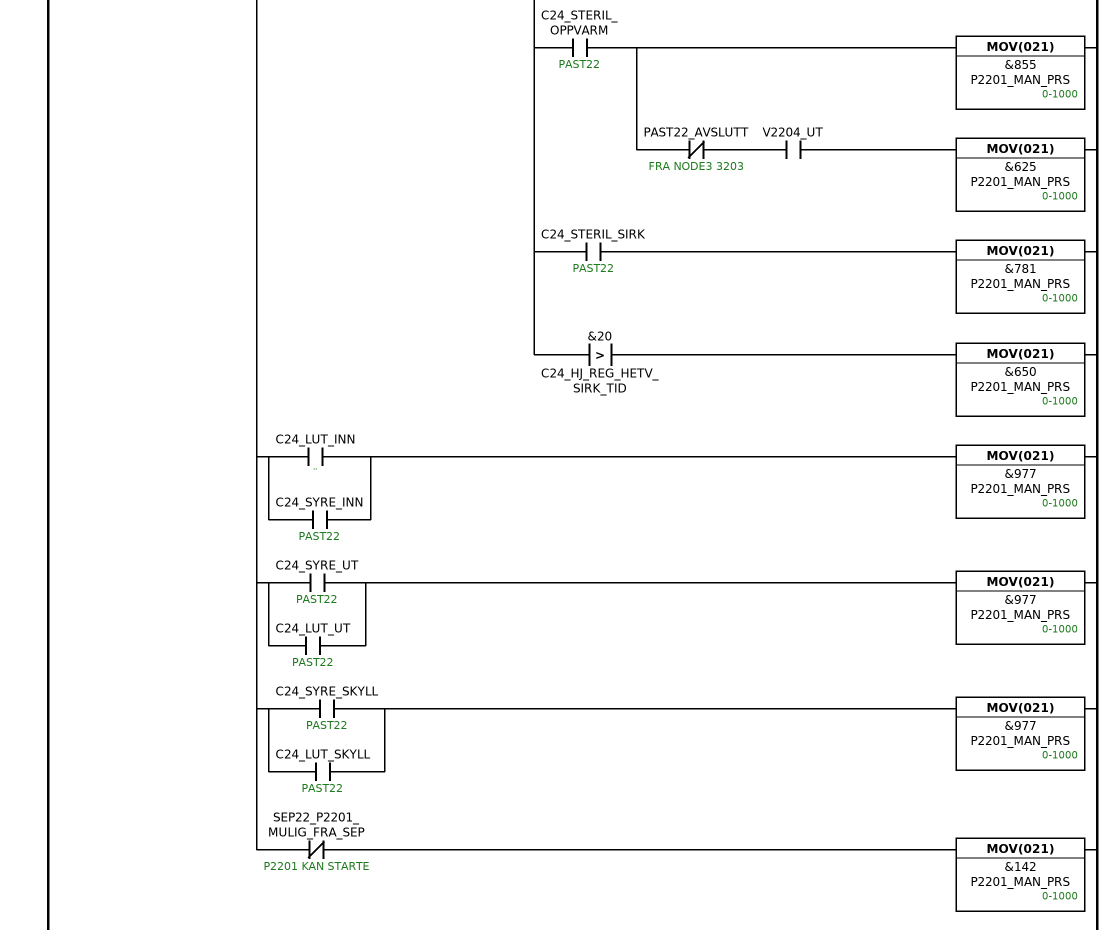
; [picture p1176: NewProgram1 / P2201, rungs 5-5]
; rung 5: REGULATOR P2201 MANUELT SETPUNKT I 0-1000
LD P_On
OUT TR0
ANDNOT PGM504_IND_C24  ; VASK PAST22
OUT TR1
AND SEP22_PART_SKUDD_INNE_FRA_SEP  ; SEP22 PARTIALSKUDD
ANDNOT 915.08
MOV(021) &590 P2201_MAN_PRS  ; 0-1000
LD TR1
AND 915.08
MOV(021) &0 P2201_MAN_PRS  ; 0-1000
LD TR0
AND PGM504_IND_C24  ; VASK PAST22
OUT TR0
@AND SEP22_PART_SKUDD_INNE_FRA_SEP  ; SEP22 PARTIALSKUDD
MOV(021) &590 P2201_MAN_PRS  ; 0-1000
LD TR0
@AND SEP22_TOT_SKUDD_INNE_FRA_SEP  ; SEP22 TOTALSKUDD(VASK)
OUT TR1
AND C24_FORSKYLL  ; PAST22
MOV(021) &448 P2201_MAN_PRS  ; 0-1000
LD TR1
AND C24_SYRE_SIRK  ; PAST22
MOV(021) &448 P2201_MAN_PRS  ; 0-1000
LD TR1
AND C24_LUT_SIRK  ; PAST22
MOV(021) &448 P2201_MAN_PRS  ; 0-1000
LD TR0
ANDNOT SEP22_PART_SKUDD_INNE_FRA_SEP  ; SEP22 PARTIALSKUDD
ANDNOT SEP22_TOT_SKUDD_INNE_FRA_SEP  ; SEP22 TOTALSKUDD(VASK)
OUT TR1
MOV(021) &977 P2201_MAN_PRS  ; 0-1000
ANDNOT PAST22_AVSLUTT  ; FRA NODE3 3203
AND V2204_UT
MOV(021) &977 P2201_MAN_PRS  ; 0-1000
LD TR1
AND C24_FORSKYLL  ; PAST22
MOV(021) &977 P2201_MAN_PRS  ; 0-1000
LD TR1
LD C24_SYRE_SIRK  ; PAST22
OR C24_LUT_SIRK  ; PAST22
ANDLD
MOV(021) &879 P2201_MAN_PRS  ; 0-1000
ANDNOT PAST22_AVSLUTT  ; FRA NODE3 3203
AND V2204_UT
MOV(021) &855 P2201_MAN_PRS  ; 0-1000
LD TR1
AND C24_STERIL_OPPVARM  ; PAST22
MOV(021) &855 P2201_MAN_PRS  ; 0-1000
ANDNOT PAST22_AVSLUTT  ; FRA NODE3 3203
AND V2204_UT
MOV(021) &625 P2201_MAN_PRS  ; 0-1000
LD TR1
AND C24_STERIL_SIRK  ; PAST22
MOV(021) &781 P2201_MAN_PRS  ; 0-1000
LD TR1
AND>(320) &20 C24_HJ_REG_HETV_SIRK_TID
MOV(021) &650 P2201_MAN_PRS  ; 0-1000
LD TR0
LD C24_LUT_INN  ; ¨
OR C24_SYRE_INN  ; PAST22
ANDLD
MOV(021) &977 P2201_MAN_PRS  ; 0-1000
LD TR0
LD C24_SYRE_UT  ; PAST22
OR C24_LUT_UT  ; PAST22
ANDLD
MOV(021) &977 P2201_MAN_PRS  ; 0-1000
LD TR0
LD C24_SYRE_SKYLL  ; PAST22
OR C24_LUT_SKYLL  ; PAST22
ANDLD
MOV(021) &977 P2201_MAN_PRS  ; 0-1000
LD TR0
ANDNOT SEP22_P2201_MULIG_FRA_SEP  ; P2201 KAN STARTE
MOV(021) &142 P2201_MAN_PRS  ; 0-1000

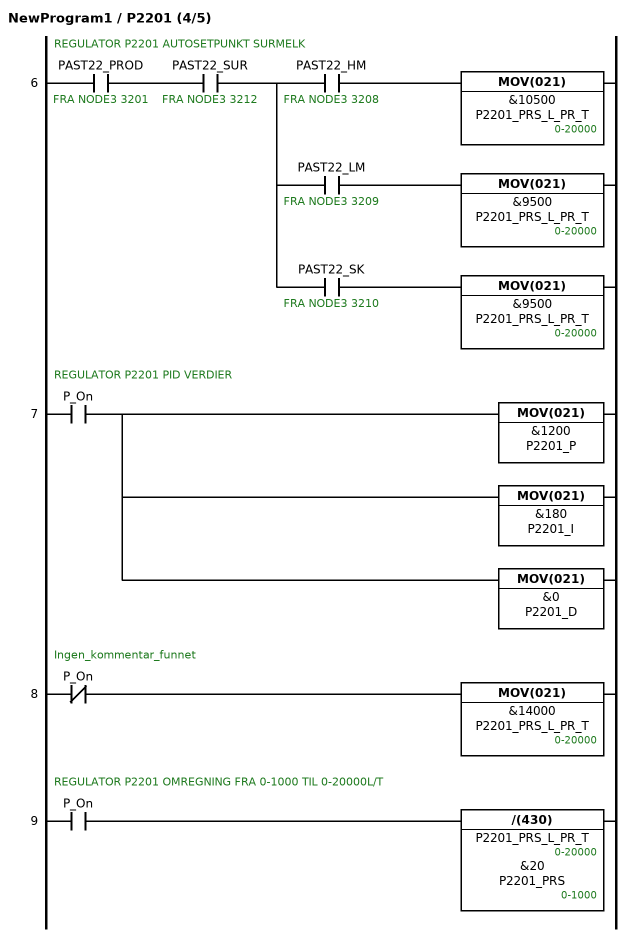
; rung 6: REGULATOR P2201 AUTOSETPUNKT SURMELK
LD PAST22_PROD  ; FRA NODE3 3201
AND PAST22_SUR  ; FRA NODE3 3212
OUT TR0
AND PAST22_HM  ; FRA NODE3 3208
MOV(021) &10500 P2201_PRS_L_PR_T  ; 0-20000
LD TR0
AND PAST22_LM  ; FRA NODE3 3209
MOV(021) &9500 P2201_PRS_L_PR_T  ; 0-20000
LD TR0
AND PAST22_SK  ; FRA NODE3 3210
MOV(021) &9500 P2201_PRS_L_PR_T  ; 0-20000
; rung 7: REGULATOR P2201 PID VERDIER
LD P_On
MOV(021) &1200 P2201_P
MOV(021) &180 P2201_I
MOV(021) &0 P2201_D
; rung 8: Ingen_kommentar_funnet
LDNOT P_On
MOV(021) &14000 P2201_PRS_L_PR_T  ; 0-20000
; rung 9: REGULATOR P2201 OMREGNING FRA 0-1000 TIL 0-20000L/T
LD P_On
/(430) P2201_PRS_L_PR_T &20 P2201_PRS  ; 0-20000, 0-1000

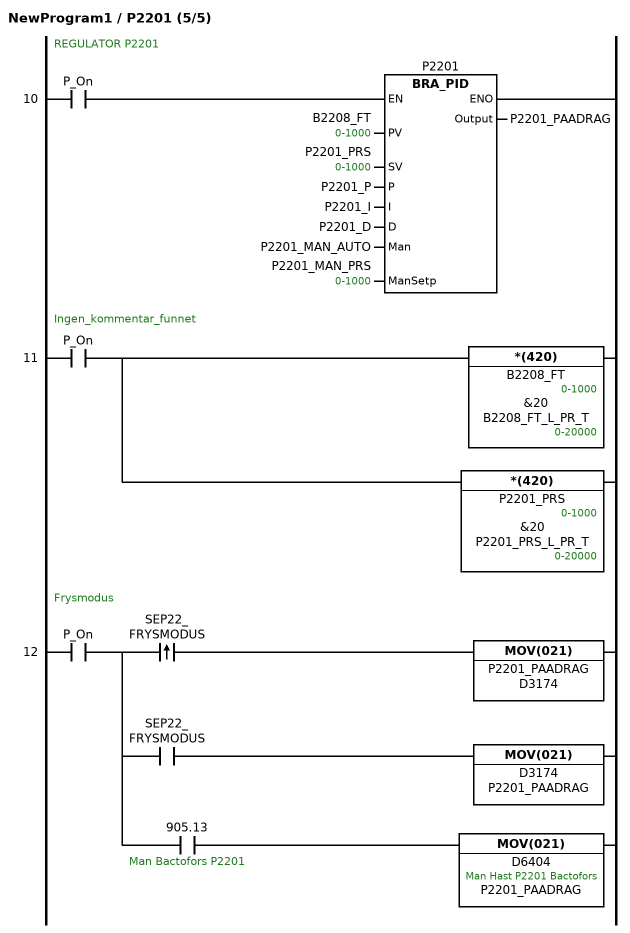
; rung 10: REGULATOR P2201
LD P_On
CALL P2201 : BRA_PID (PV := B2208_FT, SV := P2201_PRS, P := P2201_P, I := P2201_I, D := P2201_D, Man := P2201_MAN_AUTO, ManSetp := P2201_MAN_PRS, Output => P2201_PAADRAG)  ; 0-1000
; rung 11: Ingen_kommentar_funnet
LD P_On
*(420) B2208_FT &20 B2208_FT_L_PR_T  ; 0-1000, 0-20000
*(420) P2201_PRS &20 P2201_PRS_L_PR_T  ; 0-1000, 0-20000
; rung 12: Frysmodus
LD P_On
OUT TR0
@AND SEP22_FRYSMODUS
MOV(021) P2201_PAADRAG D3174
LD TR0
AND SEP22_FRYSMODUS
MOV(021) D3174 P2201_PAADRAG
LD TR0
AND 905.13  ; Man Bactofors P2201
MOV(021) D6404 P2201_PAADRAG  ; Man Hast P2201 Bactofors
; rung 13: Ingen_kommentar_funnet

### Section P2202

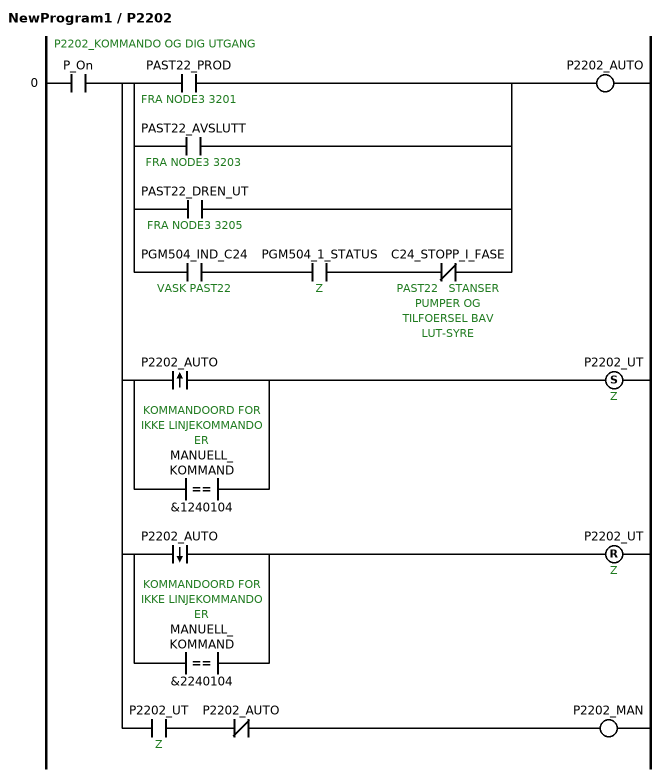
; rung 0: P2202_KOMMANDO OG DIG UTGANG
LD P_On
OUT TR0
LD PAST22_PROD  ; FRA NODE3 3201
OR PAST22_AVSLUTT  ; FRA NODE3 3203
OR PAST22_DREN_UT  ; FRA NODE3 3205
LD PGM504_IND_C24  ; VASK PAST22
AND PGM504_1_STATUS  ; Z
ANDNOT C24_STOPP_I_FASE  ; PAST22   STANSER PUMPER OG TILFOERSEL BAV LUT-SYRE
ORLD
ANDLD
OUT P2202_AUTO
LD TR0
@LD P2202_AUTO
OR=L(301) MANUELL_KOMMAND &1240104  ; KOMMANDOORD FOR IKKE LINJEKOMMANDOER
ANDLD
SET P2202_UT  ; Z
LD TR0
%LD P2202_AUTO
OR=L(301) MANUELL_KOMMAND &2240104  ; KOMMANDOORD FOR IKKE LINJEKOMMANDOER
ANDLD
RSET P2202_UT  ; Z
LD TR0
AND P2202_UT  ; Z
ANDNOT P2202_AUTO
OUT P2202_MAN
; rung 1: Ingen_kommentar_funnet

### Section P2203

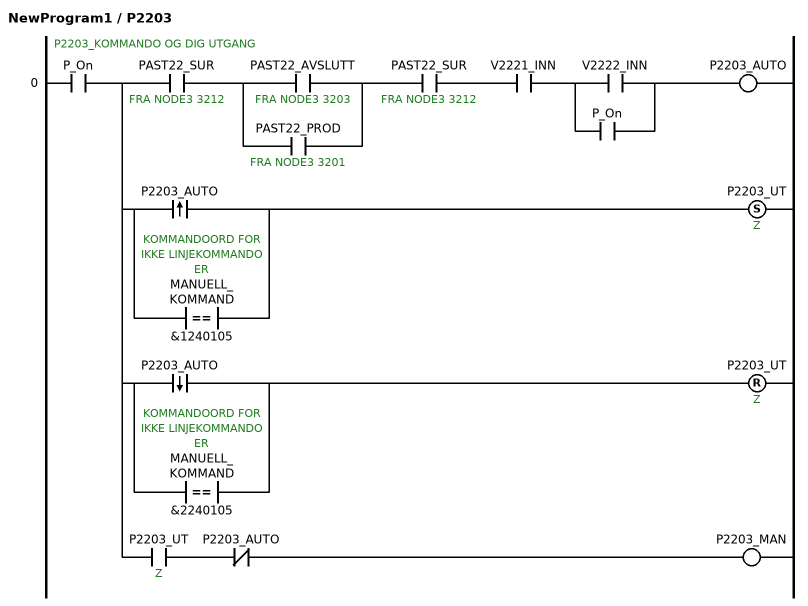
; rung 0: P2203_KOMMANDO OG DIG UTGANG
LD P_On
OUT TR0
AND PAST22_SUR  ; FRA NODE3 3212
LD PAST22_AVSLUTT  ; FRA NODE3 3203
OR PAST22_PROD  ; FRA NODE3 3201
ANDLD
AND PAST22_SUR  ; FRA NODE3 3212
AND V2221_INN
LD V2222_INN
OR P_On
ANDLD
OUT P2203_AUTO
LD TR0
@LD P2203_AUTO
OR=L(301) MANUELL_KOMMAND &1240105  ; KOMMANDOORD FOR IKKE LINJEKOMMANDOER
ANDLD
SET P2203_UT  ; Z
LD TR0
%LD P2203_AUTO
OR=L(301) MANUELL_KOMMAND &2240105  ; KOMMANDOORD FOR IKKE LINJEKOMMANDOER
ANDLD
RSET P2203_UT  ; Z
LD TR0
AND P2203_UT  ; Z
ANDNOT P2203_AUTO
OUT P2203_MAN
; rung 1: Ingen_kommentar_funnet

### Section P2204

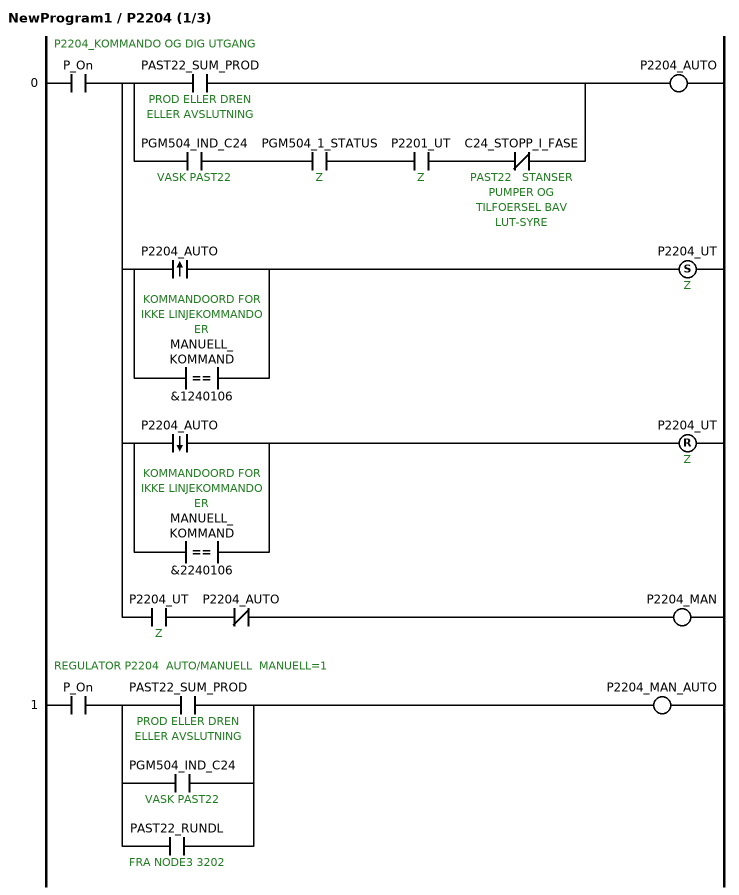
; rung 0: P2204_KOMMANDO OG DIG UTGANG
LD P_On
OUT TR0
LD PAST22_SUM_PROD  ; PROD ELLER DREN ELLER AVSLUTNING
LD PGM504_IND_C24  ; VASK PAST22
AND PGM504_1_STATUS  ; Z
AND P2201_UT  ; Z
ANDNOT C24_STOPP_I_FASE  ; PAST22   STANSER PUMPER OG TILFOERSEL BAV LUT-SYRE
ORLD
ANDLD
OUT P2204_AUTO
LD TR0
@LD P2204_AUTO
OR=L(301) MANUELL_KOMMAND &1240106  ; KOMMANDOORD FOR IKKE LINJEKOMMANDOER
ANDLD
SET P2204_UT  ; Z
LD TR0
%LD P2204_AUTO
OR=L(301) MANUELL_KOMMAND &2240106  ; KOMMANDOORD FOR IKKE LINJEKOMMANDOER
ANDLD
RSET P2204_UT  ; Z
LD TR0
AND P2204_UT  ; Z
ANDNOT P2204_AUTO
OUT P2204_MAN
; rung 1: REGULATOR P2204  AUTO/MANUELL  MANUELL=1
LD P_On
LD PAST22_SUM_PROD  ; PROD ELLER DREN ELLER AVSLUTNING
OR PGM504_IND_C24  ; VASK PAST22
OR PAST22_RUNDL  ; FRA NODE3 3202
ANDLD
OUT P2204_MAN_AUTO

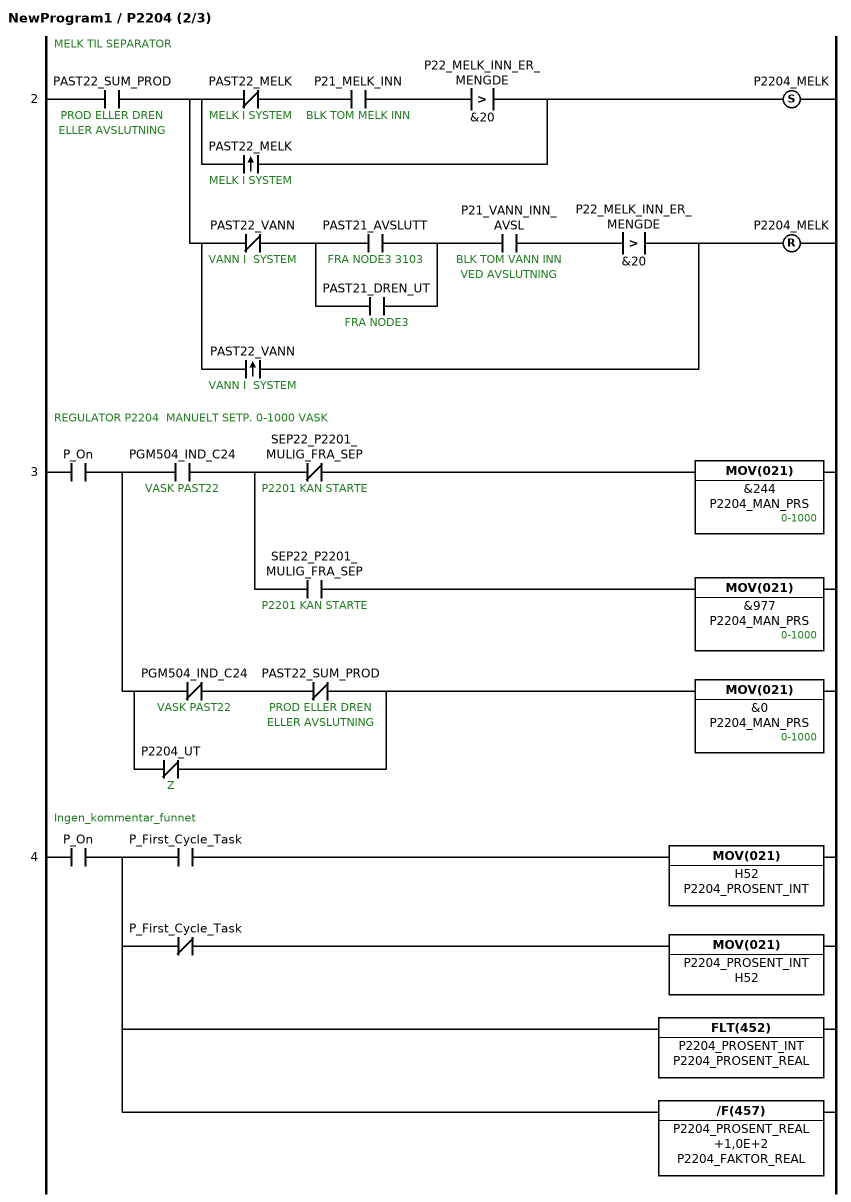
; rung 2: MELK TIL SEPARATOR
LD PAST22_SUM_PROD  ; PROD ELLER DREN ELLER AVSLUTNING
OUT TR0
LDNOT PAST22_MELK  ; MELK I SYSTEM
AND P21_MELK_INN  ; BLK TOM MELK INN
AND>L(321) P22_MELK_INN_ER_MENGDE &20
@OR PAST22_MELK  ; MELK I SYSTEM
ANDLD
SET P2204_MELK
LD TR0
LDNOT PAST22_VANN  ; VANN I  SYSTEM
LD PAST21_AVSLUTT  ; FRA NODE3 3103
OR PAST21_DREN_UT  ; FRA NODE3
ANDLD
AND P21_VANN_INN_AVSL  ; BLK TOM VANN INN VED AVSLUTNING
AND>L(321) P22_MELK_INN_ER_MENGDE &20
@OR PAST22_VANN  ; VANN I  SYSTEM
ANDLD
RSET P2204_MELK
; rung 3: REGULATOR P2204  MANUELT SETP. 0-1000 VASK
LD P_On
OUT TR0
AND PGM504_IND_C24  ; VASK PAST22
OUT TR1
ANDNOT SEP22_P2201_MULIG_FRA_SEP  ; P2201 KAN STARTE
MOV(021) &244 P2204_MAN_PRS  ; 0-1000
LD TR1
AND SEP22_P2201_MULIG_FRA_SEP  ; P2201 KAN STARTE
MOV(021) &977 P2204_MAN_PRS  ; 0-1000
LD TR0
LDNOT PGM504_IND_C24  ; VASK PAST22
ANDNOT PAST22_SUM_PROD  ; PROD ELLER DREN ELLER AVSLUTNING
ORNOT P2204_UT  ; Z
ANDLD
MOV(021) &0 P2204_MAN_PRS  ; 0-1000
; rung 4: Ingen_kommentar_funnet
LD P_On
OUT TR0
AND P_First_Cycle_Task
MOV(021) H52 P2204_PROSENT_INT
LD TR0
ANDNOT P_First_Cycle_Task
MOV(021) P2204_PROSENT_INT H52
LD TR0
FLT(452) P2204_PROSENT_INT P2204_PROSENT_REAL
/F(457) P2204_PROSENT_REAL +1,0E+2 P2204_FAKTOR_REAL

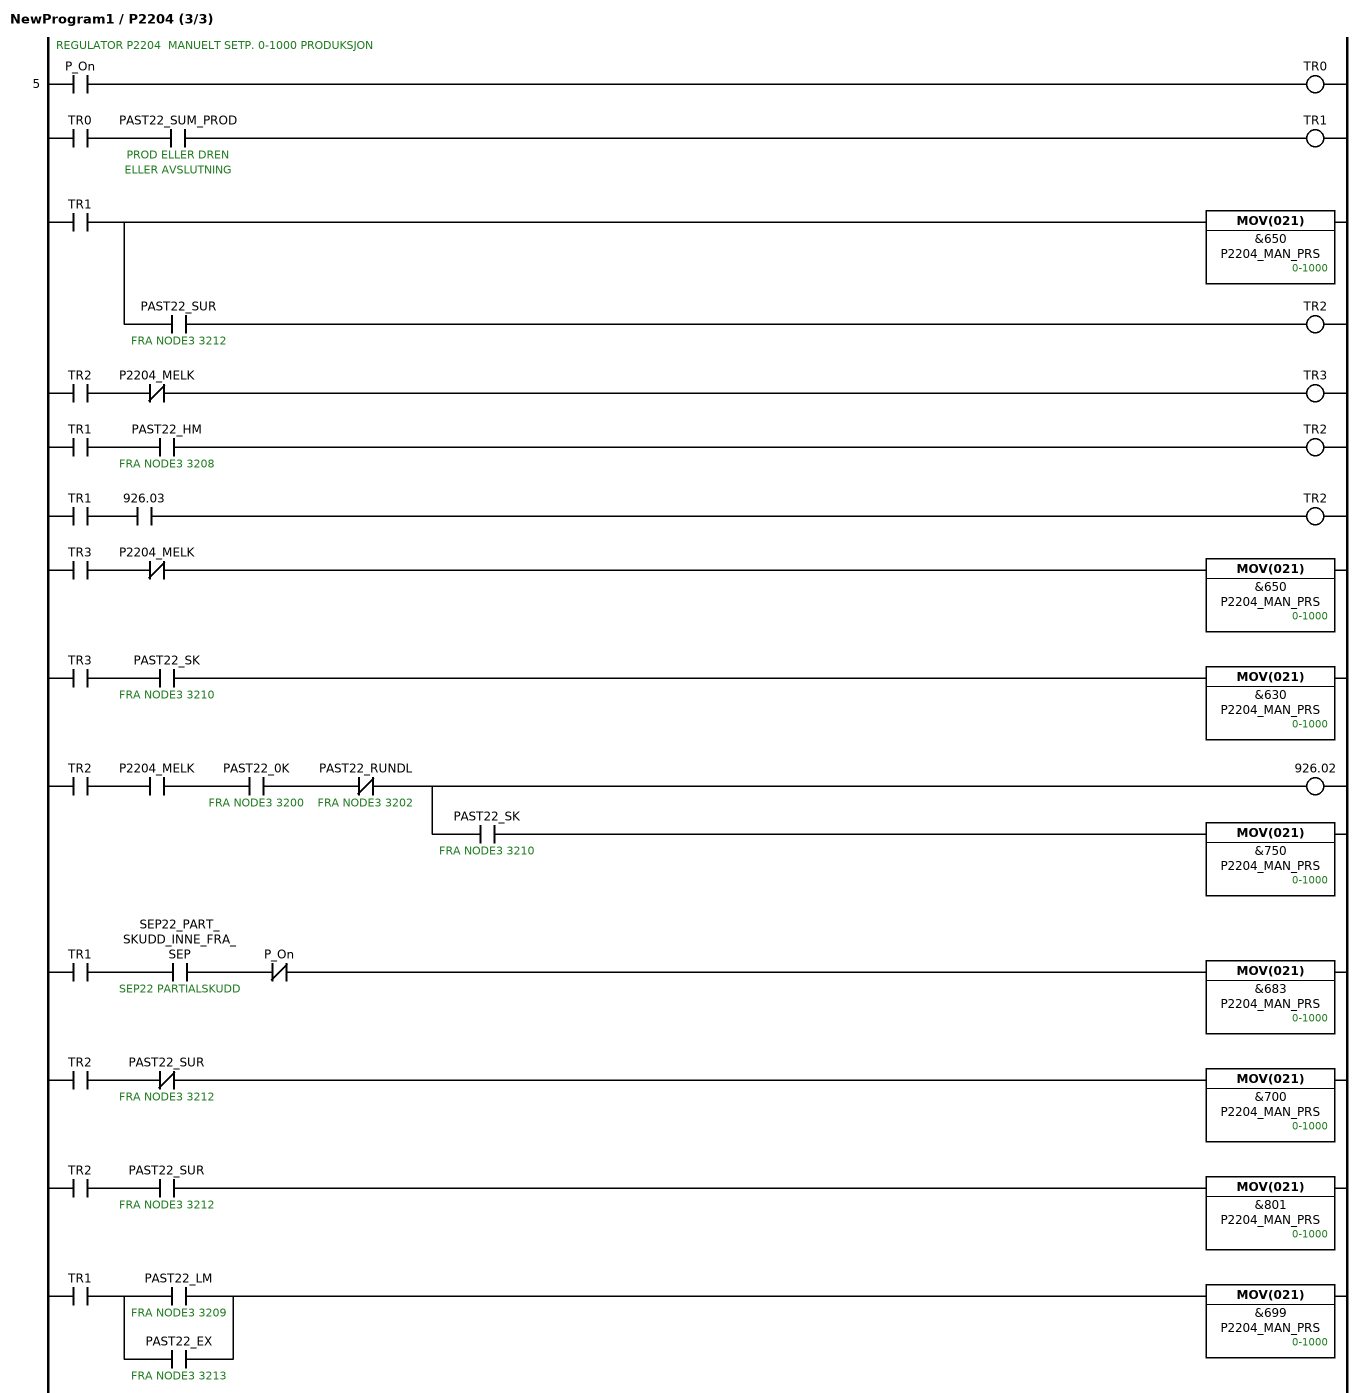

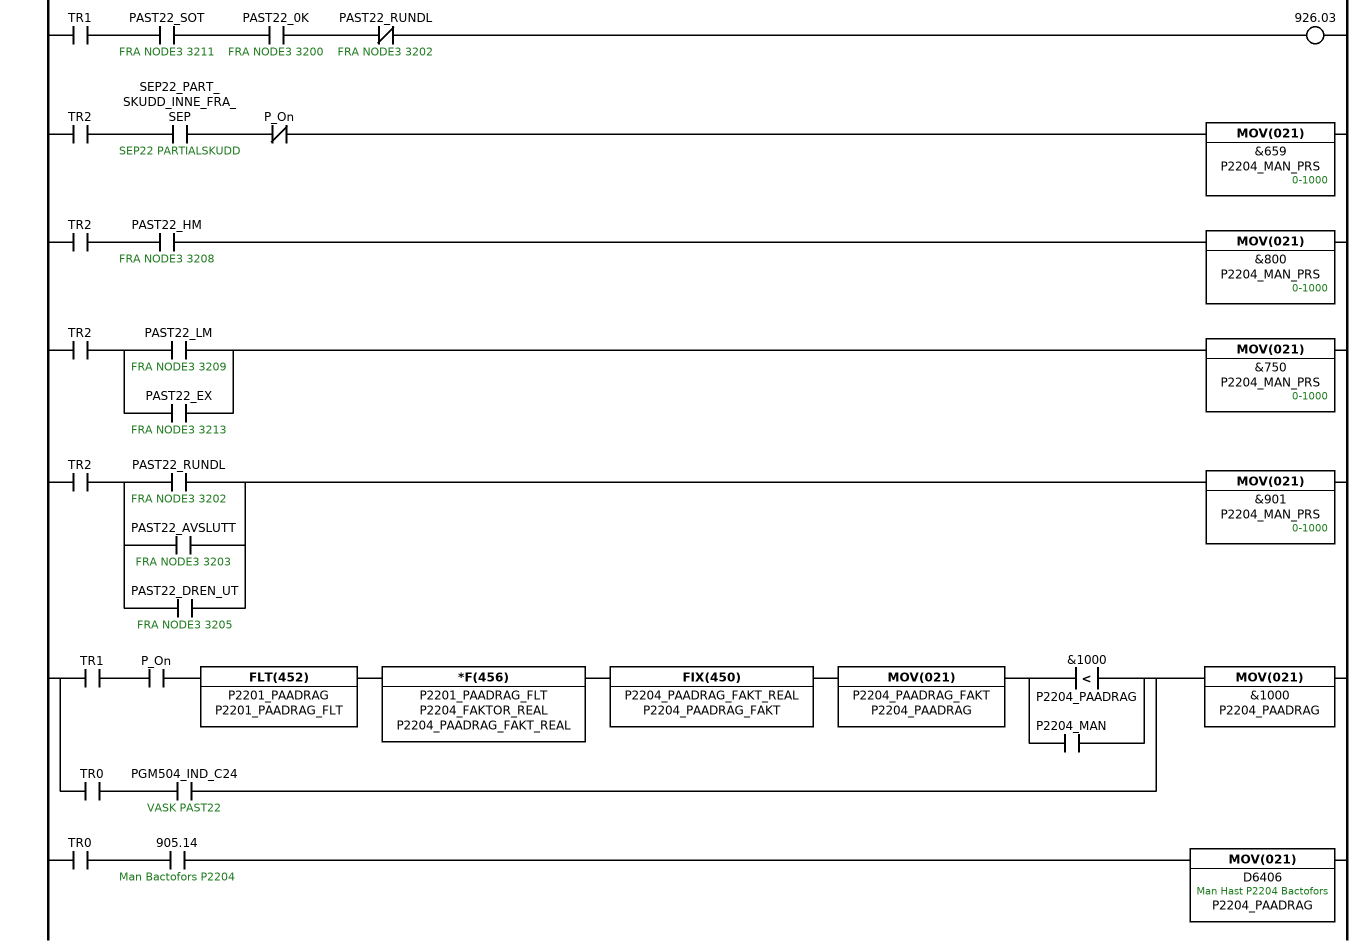
; rung 5: REGULATOR P2204  MANUELT SETP. 0-1000 PRODUKSJON
LD P_On
OUT TR0
AND PAST22_SUM_PROD  ; PROD ELLER DREN ELLER AVSLUTNING
OUT TR1
MOV(021) &650 P2204_MAN_PRS  ; 0-1000
AND PAST22_SUR  ; FRA NODE3 3212
OUT TR2
ANDNOT P2204_MELK
OUT TR3
ANDNOT P2204_MELK
MOV(021) &650 P2204_MAN_PRS  ; 0-1000
LD TR3
AND PAST22_SK  ; FRA NODE3 3210
MOV(021) &630 P2204_MAN_PRS  ; 0-1000
LD TR2
AND P2204_MELK
AND PAST22_0K  ; FRA NODE3 3200
ANDNOT PAST22_RUNDL  ; FRA NODE3 3202
OUT 926.02
AND PAST22_SK  ; FRA NODE3 3210
MOV(021) &750 P2204_MAN_PRS  ; 0-1000
LD TR1
AND SEP22_PART_SKUDD_INNE_FRA_SEP  ; SEP22 PARTIALSKUDD
ANDNOT P_On
MOV(021) &683 P2204_MAN_PRS  ; 0-1000
LD TR1
AND PAST22_HM  ; FRA NODE3 3208
OUT TR2
ANDNOT PAST22_SUR  ; FRA NODE3 3212
MOV(021) &700 P2204_MAN_PRS  ; 0-1000
LD TR2
AND PAST22_SUR  ; FRA NODE3 3212
MOV(021) &801 P2204_MAN_PRS  ; 0-1000
LD TR1
LD PAST22_LM  ; FRA NODE3 3209
OR PAST22_EX  ; FRA NODE3 3213
ANDLD
MOV(021) &699 P2204_MAN_PRS  ; 0-1000
LD TR1
AND PAST22_SOT  ; FRA NODE3 3211
AND PAST22_0K  ; FRA NODE3 3200
ANDNOT PAST22_RUNDL  ; FRA NODE3 3202
OUT 926.03
LD TR1
AND 926.03
OUT TR2
AND SEP22_PART_SKUDD_INNE_FRA_SEP  ; SEP22 PARTIALSKUDD
ANDNOT P_On
MOV(021) &659 P2204_MAN_PRS  ; 0-1000
LD TR2
AND PAST22_HM  ; FRA NODE3 3208
MOV(021) &800 P2204_MAN_PRS  ; 0-1000
LD TR2
LD PAST22_LM  ; FRA NODE3 3209
OR PAST22_EX  ; FRA NODE3 3213
ANDLD
MOV(021) &750 P2204_MAN_PRS  ; 0-1000
LD TR2
LD PAST22_RUNDL  ; FRA NODE3 3202
OR PAST22_AVSLUTT  ; FRA NODE3 3203
OR PAST22_DREN_UT  ; FRA NODE3 3205
ANDLD
MOV(021) &901 P2204_MAN_PRS  ; 0-1000
LD TR1
AND P_On
FLT(452) P2201_PAADRAG P2201_PAADRAG_FLT
*F(456) P2201_PAADRAG_FLT P2204_FAKTOR_REAL P2204_PAADRAG_FAKT_REAL
FIX(450) P2204_PAADRAG_FAKT_REAL P2204_PAADRAG_FAKT
MOV(021) P2204_PAADRAG_FAKT P2204_PAADRAG
LD<(310) &1000 P2204_PAADRAG
OR P2204_MAN
ANDLD
LD TR0
AND PGM504_IND_C24  ; VASK PAST22
ORLD
MOV(021) &1000 P2204_PAADRAG
LD TR0
AND 905.14  ; Man Bactofors P2204
MOV(021) D6406 P2204_PAADRAG  ; Man Hast P2204 Bactofors
; rung 6: Ingen_kommentar_funnet

### Section V2219

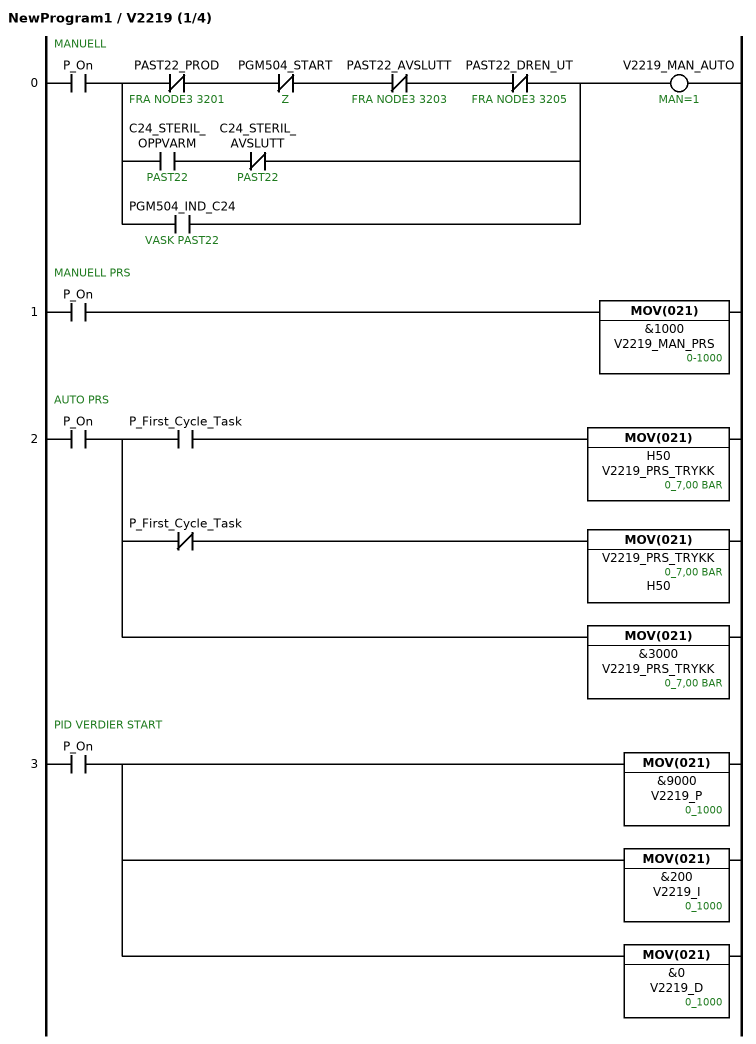
; rung 0: MANUELL
LD P_On
LDNOT PAST22_PROD  ; FRA NODE3 3201
ANDNOT PGM504_START  ; Z
ANDNOT PAST22_AVSLUTT  ; FRA NODE3 3203
ANDNOT PAST22_DREN_UT  ; FRA NODE3 3205
LD C24_STERIL_OPPVARM  ; PAST22
ANDNOT C24_STERIL_AVSLUTT  ; PAST22
ORLD
OR PGM504_IND_C24  ; VASK PAST22
ANDLD
OUT V2219_MAN_AUTO  ; MAN=1
; rung 1: MANUELL PRS
LD P_On
MOV(021) &1000 V2219_MAN_PRS  ; 0-1000
; rung 2: AUTO PRS
LD P_On
OUT TR0
AND P_First_Cycle_Task
MOV(021) H50 V2219_PRS_TRYKK  ; 0_7,00 BAR
LD TR0
ANDNOT P_First_Cycle_Task
MOV(021) V2219_PRS_TRYKK H50  ; 0_7,00 BAR
LD TR0
MOV(021) &3000 V2219_PRS_TRYKK  ; 0_7,00 BAR
; rung 3: PID VERDIER START
LD P_On
MOV(021) &9000 V2219_P  ; 0_1000
MOV(021) &200 V2219_I  ; 0_1000
MOV(021) &0 V2219_D  ; 0_1000

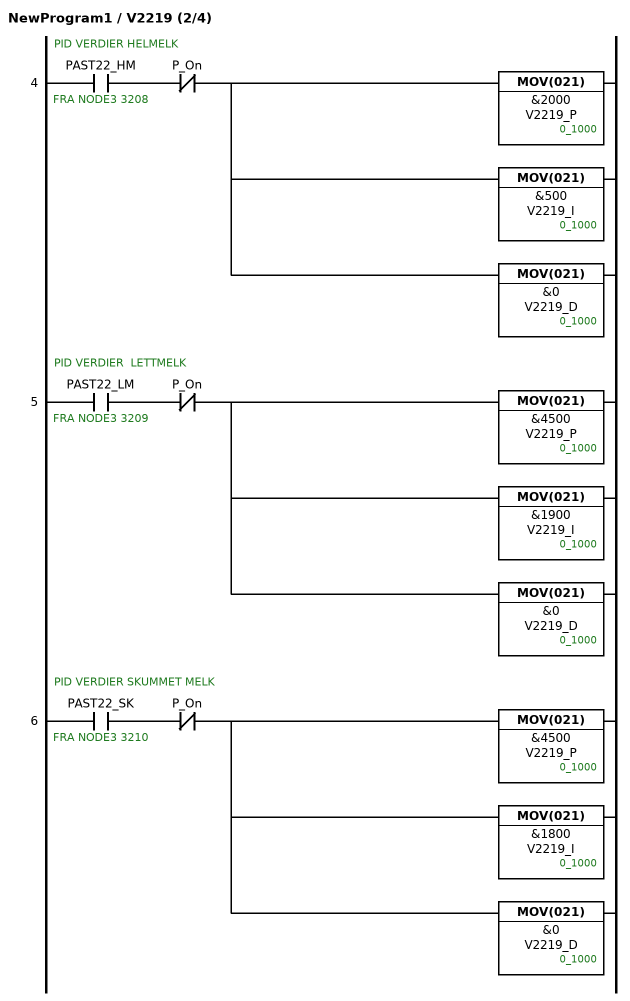
; rung 4: PID VERDIER HELMELK
LD PAST22_HM  ; FRA NODE3 3208
ANDNOT P_On
MOV(021) &2000 V2219_P  ; 0_1000
MOV(021) &500 V2219_I  ; 0_1000
MOV(021) &0 V2219_D  ; 0_1000
; rung 5: PID VERDIER  LETTMELK
LD PAST22_LM  ; FRA NODE3 3209
ANDNOT P_On
MOV(021) &4500 V2219_P  ; 0_1000
MOV(021) &1900 V2219_I  ; 0_1000
MOV(021) &0 V2219_D  ; 0_1000
; rung 6: PID VERDIER SKUMMET MELK
LD PAST22_SK  ; FRA NODE3 3210
ANDNOT P_On
MOV(021) &4500 V2219_P  ; 0_1000
MOV(021) &1800 V2219_I  ; 0_1000
MOV(021) &0 V2219_D  ; 0_1000

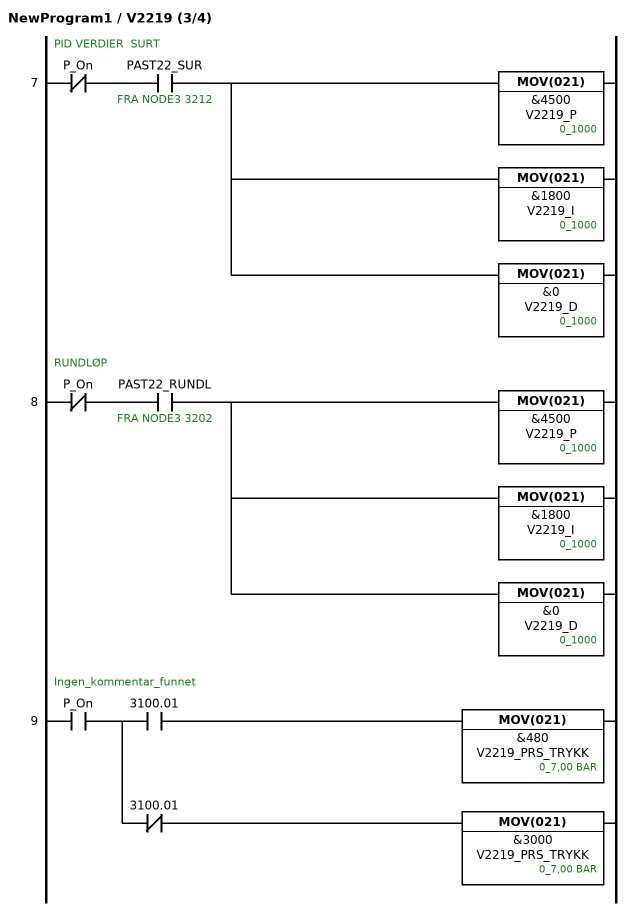
; rung 7: PID VERDIER  SURT
LDNOT P_On
AND PAST22_SUR  ; FRA NODE3 3212
MOV(021) &4500 V2219_P  ; 0_1000
MOV(021) &1800 V2219_I  ; 0_1000
MOV(021) &0 V2219_D  ; 0_1000
; rung 8: RUNDLØP
LDNOT P_On
AND PAST22_RUNDL  ; FRA NODE3 3202
MOV(021) &4500 V2219_P  ; 0_1000
MOV(021) &1800 V2219_I  ; 0_1000
MOV(021) &0 V2219_D  ; 0_1000
; rung 9: Ingen_kommentar_funnet
LD P_On
OUT TR0
AND 3100.01
MOV(021) &480 V2219_PRS_TRYKK  ; 0_7,00 BAR
LD TR0
ANDNOT 3100.01
MOV(021) &3000 V2219_PRS_TRYKK  ; 0_7,00 BAR

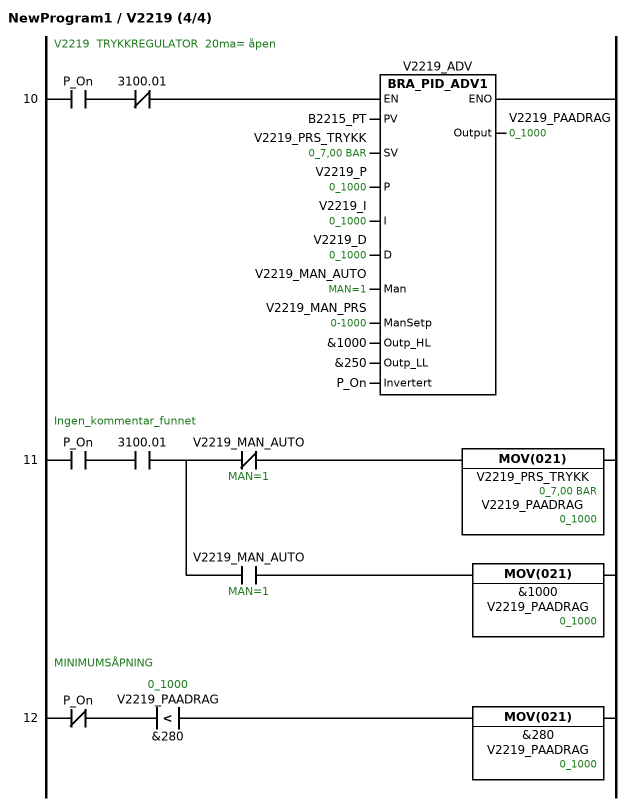
; rung 10: V2219  TRYKKREGULATOR  20ma= åpen
LD P_On
ANDNOT 3100.01
CALL V2219_ADV : BRA_PID_ADV1 (PV := B2215_PT, SV := V2219_PRS_TRYKK, P := V2219_P, I := V2219_I, D := V2219_D, Man := V2219_MAN_AUTO, ManSetp := V2219_MAN_PRS, Outp_HL := &1000, Outp_LL := &250, Invertert := P_On, Output => V2219_PAADRAG)  ; 0_7,00 BAR, 0_1000, MAN=1, 0-1000
; rung 11: Ingen_kommentar_funnet
LD P_On
AND 3100.01
OUT TR0
ANDNOT V2219_MAN_AUTO  ; MAN=1
MOV(021) V2219_PRS_TRYKK V2219_PAADRAG  ; 0_7,00 BAR, 0_1000
LD TR0
AND V2219_MAN_AUTO  ; MAN=1
MOV(021) &1000 V2219_PAADRAG  ; 0_1000
; rung 12: MINIMUMSÅPNING
LDNOT P_On
AND<(310) V2219_PAADRAG &280  ; 0_1000
MOV(021) &280 V2219_PAADRAG  ; 0_1000
; rung 13: Ingen_kommentar_funnet

### Section V2252

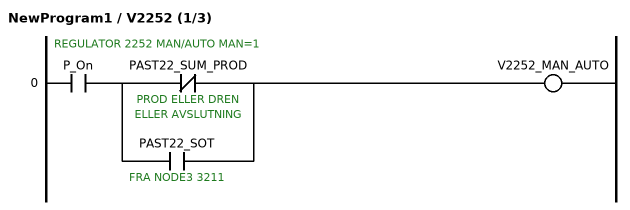
; rung 0: REGULATOR 2252 MAN/AUTO MAN=1
LD P_On
LDNOT PAST22_SUM_PROD  ; PROD ELLER DREN ELLER AVSLUTNING
OR PAST22_SOT  ; FRA NODE3 3211
ANDLD
OUT V2252_MAN_AUTO

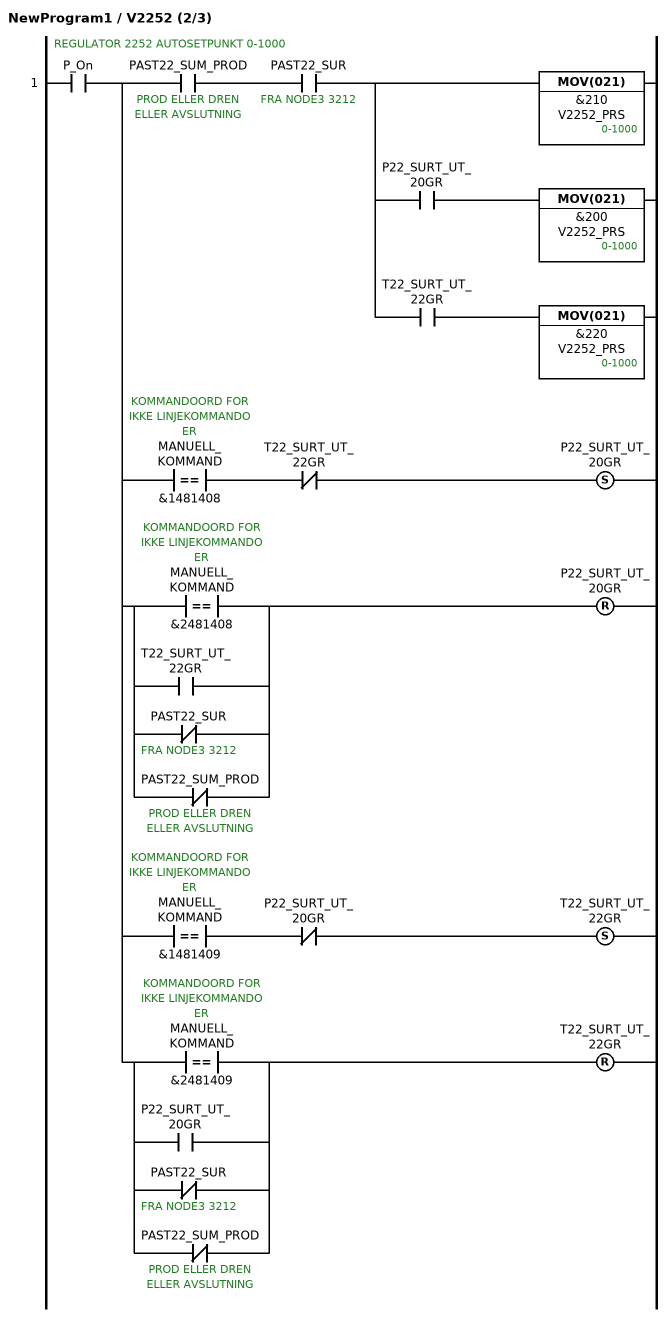
; rung 1: REGULATOR 2252 AUTOSETPUNKT 0-1000
LD P_On
OUT TR0
AND PAST22_SUM_PROD  ; PROD ELLER DREN ELLER AVSLUTNING
AND PAST22_SUR  ; FRA NODE3 3212
OUT TR1
MOV(021) &210 V2252_PRS  ; 0-1000
AND P22_SURT_UT_20GR
MOV(021) &200 V2252_PRS  ; 0-1000
LD TR1
AND T22_SURT_UT_22GR
MOV(021) &220 V2252_PRS  ; 0-1000
LD TR0
AND=L(301) MANUELL_KOMMAND &1481408  ; KOMMANDOORD FOR IKKE LINJEKOMMANDOER
ANDNOT T22_SURT_UT_22GR
SET P22_SURT_UT_20GR
LD TR0
LD=L(301) MANUELL_KOMMAND &2481408  ; KOMMANDOORD FOR IKKE LINJEKOMMANDOER
OR T22_SURT_UT_22GR
ORNOT PAST22_SUR  ; FRA NODE3 3212
ORNOT PAST22_SUM_PROD  ; PROD ELLER DREN ELLER AVSLUTNING
ANDLD
RSET P22_SURT_UT_20GR
LD TR0
AND=L(301) MANUELL_KOMMAND &1481409  ; KOMMANDOORD FOR IKKE LINJEKOMMANDOER
ANDNOT P22_SURT_UT_20GR
SET T22_SURT_UT_22GR
LD TR0
LD=L(301) MANUELL_KOMMAND &2481409  ; KOMMANDOORD FOR IKKE LINJEKOMMANDOER
OR P22_SURT_UT_20GR
ORNOT PAST22_SUR  ; FRA NODE3 3212
ORNOT PAST22_SUM_PROD  ; PROD ELLER DREN ELLER AVSLUTNING
ANDLD
RSET T22_SURT_UT_22GR

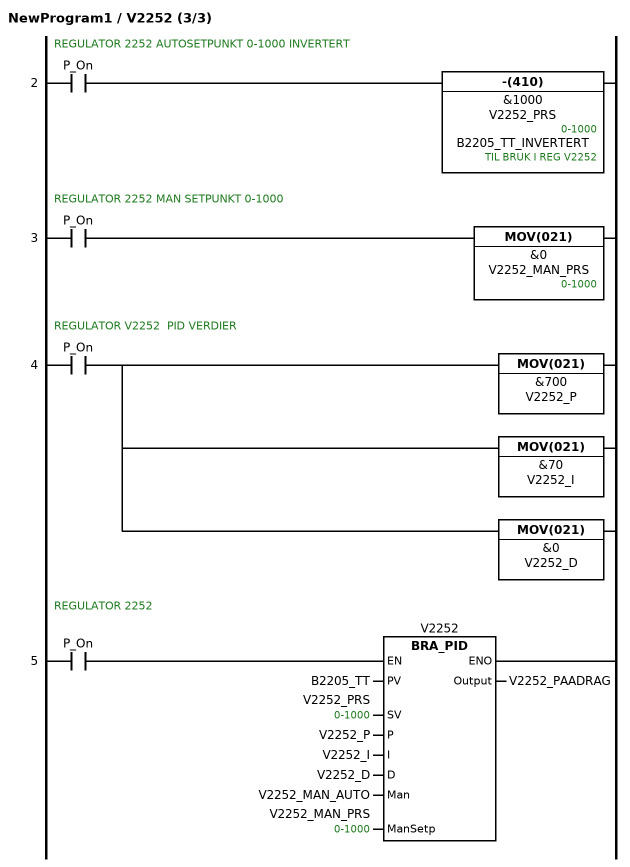
; rung 2: REGULATOR 2252 AUTOSETPUNKT 0-1000 INVERTERT
LD P_On
-(410) &1000 V2252_PRS B2205_TT_INVERTERT  ; 0-1000, TIL BRUK I REG V2252
; rung 3: REGULATOR 2252 MAN SETPUNKT 0-1000
LD P_On
MOV(021) &0 V2252_MAN_PRS  ; 0-1000
; rung 4: REGULATOR V2252  PID VERDIER
LD P_On
MOV(021) &700 V2252_P
MOV(021) &70 V2252_I
MOV(021) &0 V2252_D
; rung 5: REGULATOR 2252
LD P_On
CALL V2252 : BRA_PID (PV := B2205_TT, SV := V2252_PRS, P := V2252_P, I := V2252_I, D := V2252_D, Man := V2252_MAN_AUTO, ManSetp := V2252_MAN_PRS, Output => V2252_PAADRAG)  ; 0-1000
; rung 6: Ingen_kommentar_funnet

### Section V2261

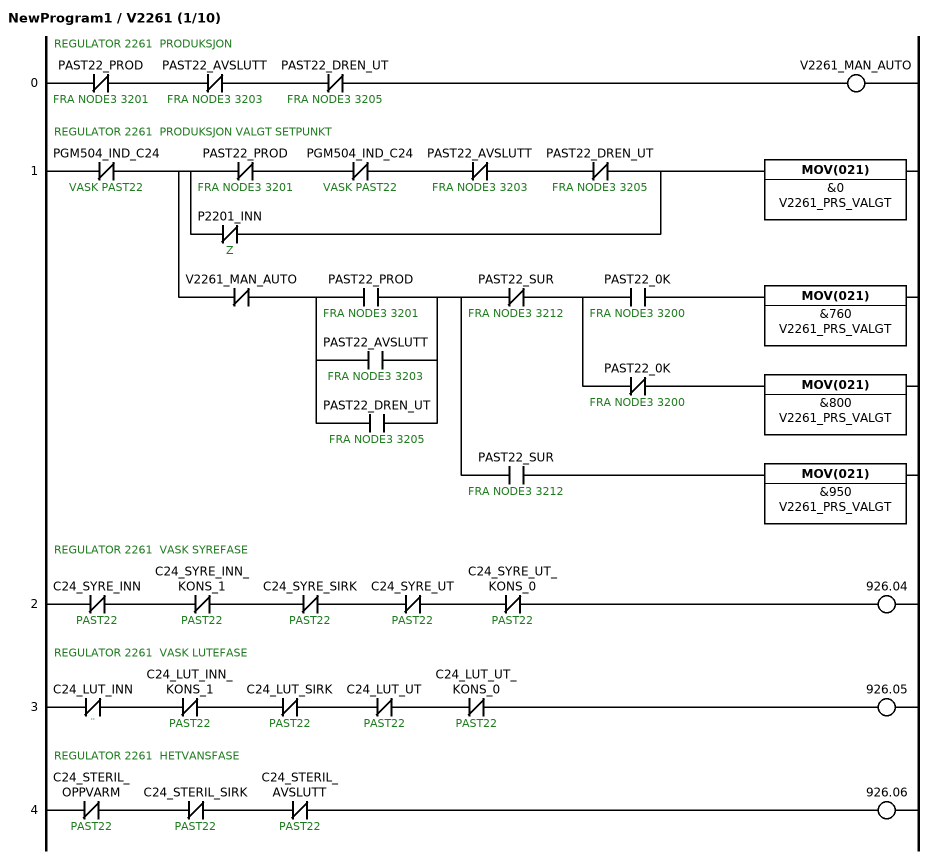
; rung 0: REGULATOR 2261  PRODUKSJON
LDNOT PAST22_PROD  ; FRA NODE3 3201
ANDNOT PAST22_AVSLUTT  ; FRA NODE3 3203
ANDNOT PAST22_DREN_UT  ; FRA NODE3 3205
OUT V2261_MAN_AUTO
; rung 1: REGULATOR 2261  PRODUKSJON VALGT SETPUNKT
LDNOT PGM504_IND_C24  ; VASK PAST22
OUT TR0
LDNOT PAST22_PROD  ; FRA NODE3 3201
ANDNOT PGM504_IND_C24  ; VASK PAST22
ANDNOT PAST22_AVSLUTT  ; FRA NODE3 3203
ANDNOT PAST22_DREN_UT  ; FRA NODE3 3205
ORNOT P2201_INN  ; Z
ANDLD
MOV(021) &0 V2261_PRS_VALGT
LD TR0
ANDNOT V2261_MAN_AUTO
LD PAST22_PROD  ; FRA NODE3 3201
OR PAST22_AVSLUTT  ; FRA NODE3 3203
OR PAST22_DREN_UT  ; FRA NODE3 3205
ANDLD
OUT TR0
ANDNOT PAST22_SUR  ; FRA NODE3 3212
OUT TR1
AND PAST22_0K  ; FRA NODE3 3200
MOV(021) &760 V2261_PRS_VALGT
LD TR1
ANDNOT PAST22_0K  ; FRA NODE3 3200
MOV(021) &800 V2261_PRS_VALGT
LD TR0
AND PAST22_SUR  ; FRA NODE3 3212
MOV(021) &950 V2261_PRS_VALGT
; rung 2: REGULATOR 2261  VASK SYREFASE
LDNOT C24_SYRE_INN  ; PAST22
ANDNOT C24_SYRE_INN_KONS_1  ; PAST22
ANDNOT C24_SYRE_SIRK  ; PAST22
ANDNOT C24_SYRE_UT  ; PAST22
ANDNOT C24_SYRE_UT_KONS_0  ; PAST22
OUT 926.04
; rung 3: REGULATOR 2261  VASK LUTEFASE
LDNOT C24_LUT_INN  ; ¨
ANDNOT C24_LUT_INN_KONS_1  ; PAST22
ANDNOT C24_LUT_SIRK  ; PAST22
ANDNOT C24_LUT_UT  ; PAST22
ANDNOT C24_LUT_UT_KONS_0  ; PAST22
OUT 926.05
; rung 4: REGULATOR 2261  HETVANSFASE
LDNOT C24_STERIL_OPPVARM  ; PAST22
ANDNOT C24_STERIL_SIRK  ; PAST22
ANDNOT C24_STERIL_AVSLUTT  ; PAST22
OUT 926.06

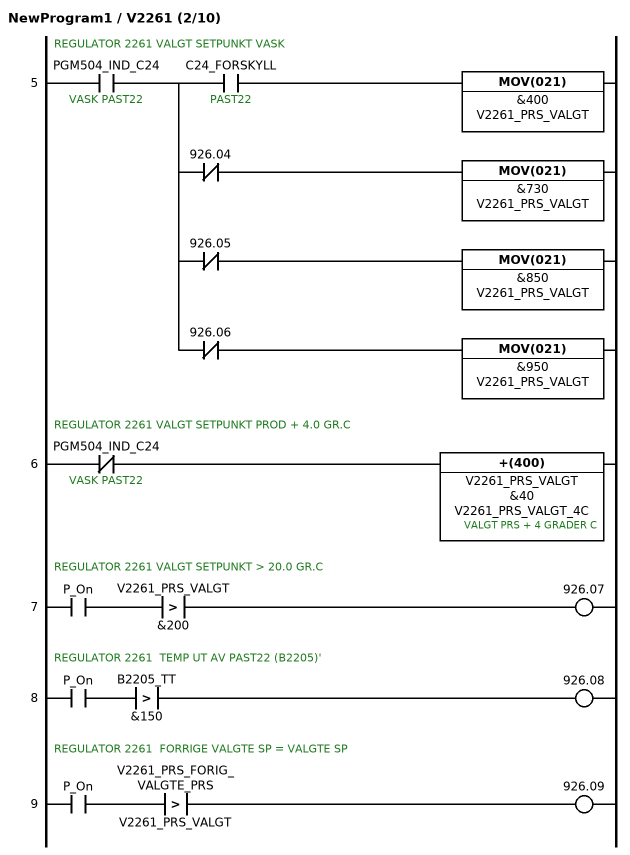
; rung 5: REGULATOR 2261 VALGT SETPUNKT VASK
LD PGM504_IND_C24  ; VASK PAST22
OUT TR0
AND C24_FORSKYLL  ; PAST22
MOV(021) &400 V2261_PRS_VALGT
LD TR0
ANDNOT 926.04
MOV(021) &730 V2261_PRS_VALGT
LD TR0
ANDNOT 926.05
MOV(021) &850 V2261_PRS_VALGT
LD TR0
ANDNOT 926.06
MOV(021) &950 V2261_PRS_VALGT
; rung 6: REGULATOR 2261 VALGT SETPUNKT PROD + 4.0 GR.C
LDNOT PGM504_IND_C24  ; VASK PAST22
+(400) V2261_PRS_VALGT &40 V2261_PRS_VALGT_4C  ; VALGT PRS + 4 GRADER C
; rung 7: REGULATOR 2261 VALGT SETPUNKT > 20.0 GR.C
LD P_On
AND>(320) V2261_PRS_VALGT &200
OUT 926.07
; rung 8: REGULATOR 2261  TEMP UT AV PAST22 (B2205)'
LD P_On
AND>(320) B2205_TT &150
OUT 926.08
; rung 9: REGULATOR 2261  FORRIGE VALGTE SP = VALGTE SP
LD P_On
AND>(320) V2261_PRS_FORIG_VALGTE_PRS V2261_PRS_VALGT
OUT 926.09

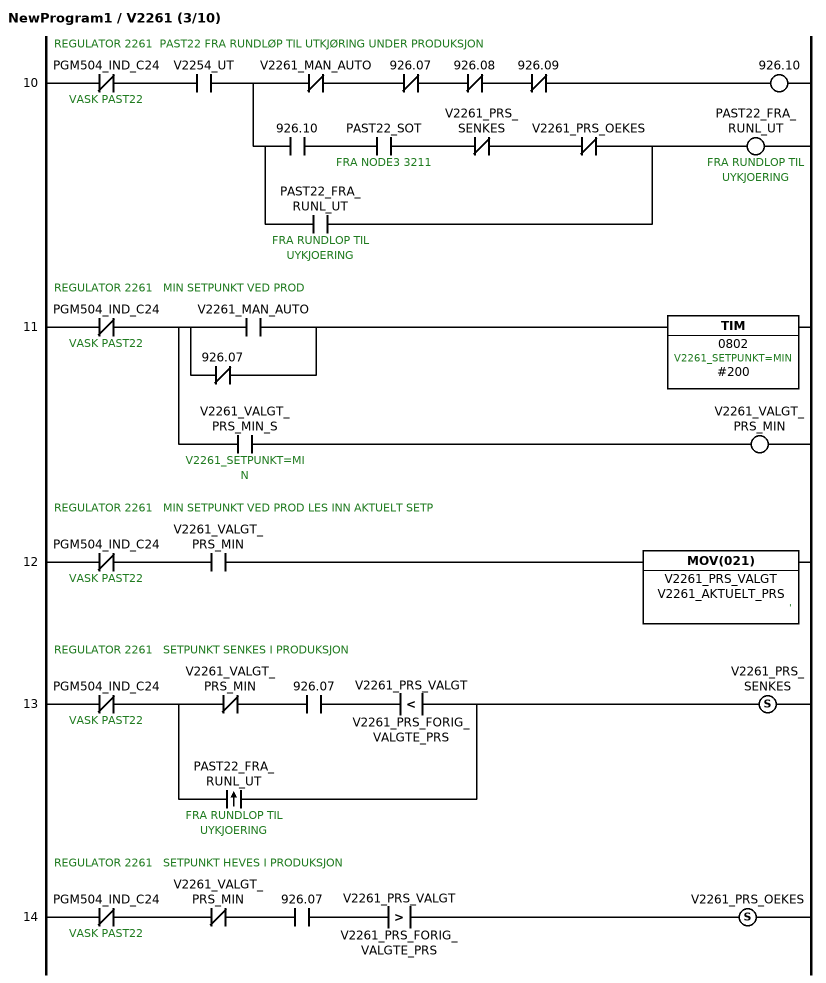
; rung 10: REGULATOR 2261  PAST22 FRA RUNDLØP TIL UTKJØRING UNDER PRODUKSJON
LDNOT PGM504_IND_C24  ; VASK PAST22
AND V2254_UT
OUT TR0
ANDNOT V2261_MAN_AUTO
ANDNOT 926.07
ANDNOT 926.08
ANDNOT 926.09
OUT 926.10
LD TR0
LD 926.10
AND PAST22_SOT  ; FRA NODE3 3211
ANDNOT V2261_PRS_SENKES
ANDNOT V2261_PRS_OEKES
OR PAST22_FRA_RUNL_UT  ; FRA RUNDLOP TIL UYKJOERING
ANDLD
OUT PAST22_FRA_RUNL_UT  ; FRA RUNDLOP TIL UYKJOERING
; rung 11: REGULATOR 2261   MIN SETPUNKT VED PROD
LDNOT PGM504_IND_C24  ; VASK PAST22
OUT TR0
LD V2261_MAN_AUTO
ORNOT 926.07
ANDLD
TIM 0802 #200  ; V2261_SETPUNKT=MIN
LD TR0
AND V2261_VALGT_PRS_MIN_S  ; V2261_SETPUNKT=MIN
OUT V2261_VALGT_PRS_MIN
; rung 12: REGULATOR 2261   MIN SETPUNKT VED PROD LES INN AKTUELT SETP
LDNOT PGM504_IND_C24  ; VASK PAST22
AND V2261_VALGT_PRS_MIN
MOV(021) V2261_PRS_VALGT V2261_AKTUELT_PRS  ; '
; rung 13: REGULATOR 2261   SETPUNKT SENKES I PRODUKSJON
LDNOT PGM504_IND_C24  ; VASK PAST22
LDNOT V2261_VALGT_PRS_MIN
AND 926.07
AND<(310) V2261_PRS_VALGT V2261_PRS_FORIG_VALGTE_PRS
@OR PAST22_FRA_RUNL_UT  ; FRA RUNDLOP TIL UYKJOERING
ANDLD
SET V2261_PRS_SENKES
; rung 14: REGULATOR 2261   SETPUNKT HEVES I PRODUKSJON
LDNOT PGM504_IND_C24  ; VASK PAST22
ANDNOT V2261_VALGT_PRS_MIN
AND 926.07
AND>(320) V2261_PRS_VALGT V2261_PRS_FORIG_VALGTE_PRS
SET V2261_PRS_OEKES

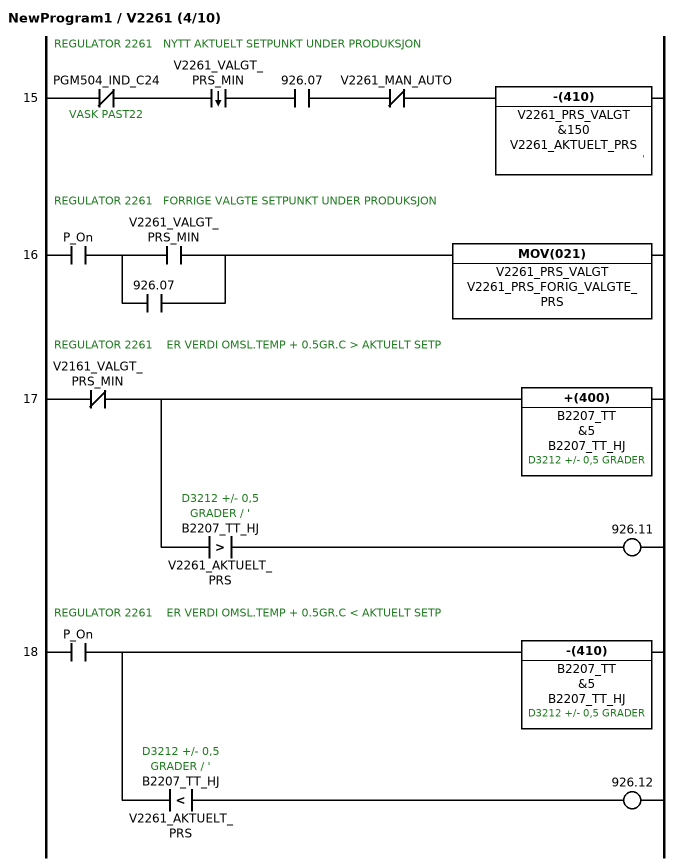
; rung 15: REGULATOR 2261   NYTT AKTUELT SETPUNKT UNDER PRODUKSJON
LDNOT PGM504_IND_C24  ; VASK PAST22
%AND V2261_VALGT_PRS_MIN
AND 926.07
ANDNOT V2261_MAN_AUTO
-(410) V2261_PRS_VALGT &150 V2261_AKTUELT_PRS  ; '
; rung 16: REGULATOR 2261   FORRIGE VALGTE SETPUNKT UNDER PRODUKSJON
LD P_On
LD V2261_VALGT_PRS_MIN
OR 926.07
ANDLD
MOV(021) V2261_PRS_VALGT V2261_PRS_FORIG_VALGTE_PRS
; rung 17: REGULATOR 2261    ER VERDI OMSL.TEMP + 0.5GR.C > AKTUELT SETP
LDNOT V2161_VALGT_PRS_MIN
+(400) B2207_TT &5 B2207_TT_HJ  ; D3212 +/- 0,5 GRADER
AND>(320) B2207_TT_HJ V2261_AKTUELT_PRS  ; D3212 +/- 0,5 GRADER, '
OUT 926.11
; rung 18: REGULATOR 2261    ER VERDI OMSL.TEMP + 0.5GR.C < AKTUELT SETP
LD P_On
-(410) B2207_TT &5 B2207_TT_HJ  ; D3212 +/- 0,5 GRADER
AND<(310) B2207_TT_HJ V2261_AKTUELT_PRS  ; D3212 +/- 0,5 GRADER, '
OUT 926.12

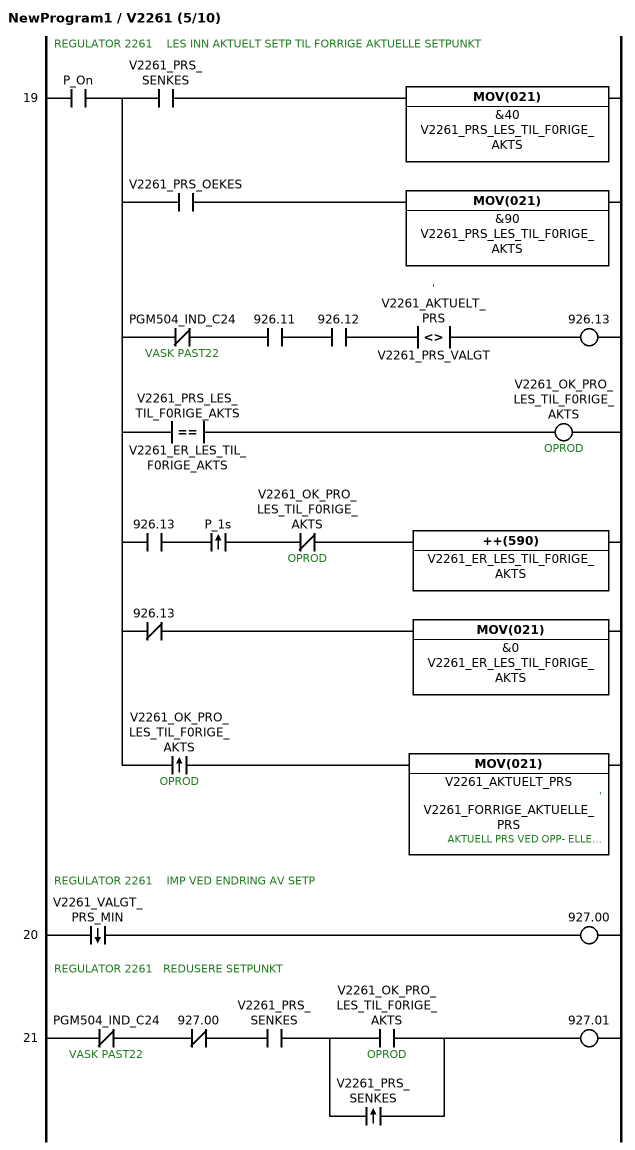
; rung 19: REGULATOR 2261    LES INN AKTUELT SETP TIL FORRIGE AKTUELLE SETPUNKT
LD P_On
OUT TR0
AND V2261_PRS_SENKES
MOV(021) &40 V2261_PRS_LES_TIL_F0RIGE_AKTS
LD TR0
AND V2261_PRS_OEKES
MOV(021) &90 V2261_PRS_LES_TIL_F0RIGE_AKTS
LD TR0
ANDNOT PGM504_IND_C24  ; VASK PAST22
AND 926.11
AND 926.12
AND<>(305) V2261_AKTUELT_PRS V2261_PRS_VALGT  ; '
OUT 926.13
LD TR0
AND=(300) V2261_PRS_LES_TIL_F0RIGE_AKTS V2261_ER_LES_TIL_F0RIGE_AKTS
OUT V2261_OK_PRO_LES_TIL_F0RIGE_AKTS  ; OPROD
LD TR0
AND 926.13
@AND P_1s
ANDNOT V2261_OK_PRO_LES_TIL_F0RIGE_AKTS  ; OPROD
++(590) V2261_ER_LES_TIL_F0RIGE_AKTS
LD TR0
ANDNOT 926.13
MOV(021) &0 V2261_ER_LES_TIL_F0RIGE_AKTS
LD TR0
@AND V2261_OK_PRO_LES_TIL_F0RIGE_AKTS  ; OPROD
MOV(021) V2261_AKTUELT_PRS V2261_FORRIGE_AKTUELLE_PRS  ; ', AKTUELL PRS VED OPP- ELLER NEDTRAPPING
; rung 20: REGULATOR 2261    IMP VED ENDRING AV SETP
%LD V2261_VALGT_PRS_MIN
OUT 927.00
; rung 21: REGULATOR 2261   REDUSERE SETPUNKT
LDNOT PGM504_IND_C24  ; VASK PAST22
ANDNOT 927.00
AND V2261_PRS_SENKES
LD V2261_OK_PRO_LES_TIL_F0RIGE_AKTS  ; OPROD
@OR V2261_PRS_SENKES
ANDLD
OUT 927.01

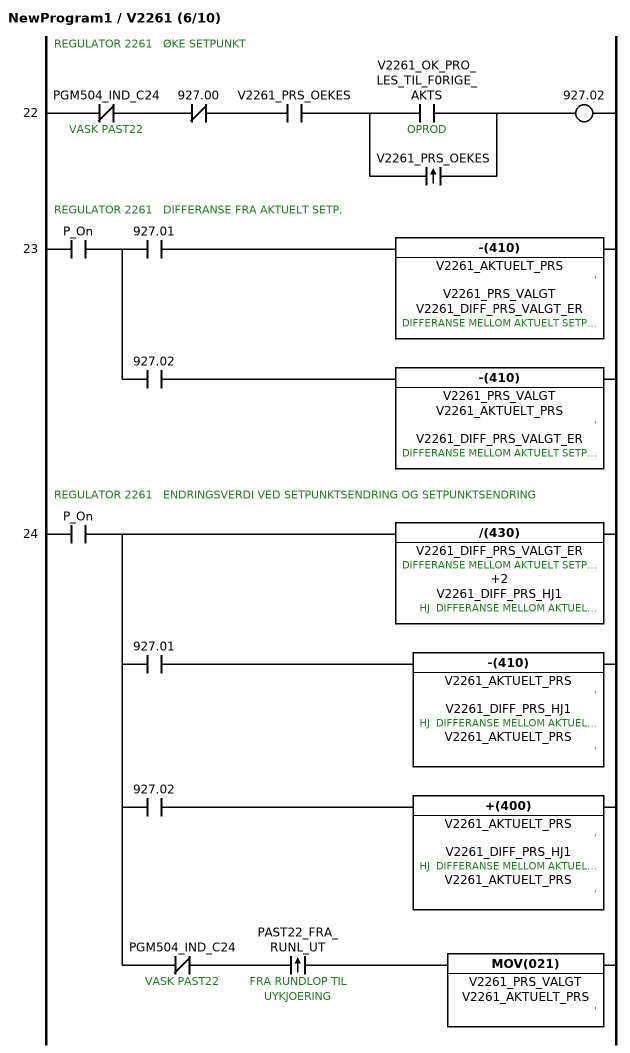
; rung 22: REGULATOR 2261   ØKE SETPUNKT
LDNOT PGM504_IND_C24  ; VASK PAST22
ANDNOT 927.00
AND V2261_PRS_OEKES
LD V2261_OK_PRO_LES_TIL_F0RIGE_AKTS  ; OPROD
@OR V2261_PRS_OEKES
ANDLD
OUT 927.02
; rung 23: REGULATOR 2261   DIFFERANSE FRA AKTUELT SETP.
LD P_On
OUT TR0
AND 927.01
-(410) V2261_AKTUELT_PRS V2261_PRS_VALGT V2261_DIFF_PRS_VALGT_ER  ; ', DIFFERANSE MELLOM AKTUELT SETP. OG VALGT SETP
LD TR0
AND 927.02
-(410) V2261_PRS_VALGT V2261_AKTUELT_PRS V2261_DIFF_PRS_VALGT_ER  ; ', DIFFERANSE MELLOM AKTUELT SETP. OG VALGT SETP
; rung 24: REGULATOR 2261   ENDRINGSVERDI VED SETPUNKTSENDRING OG SETPUNKTSENDRING
LD P_On
OUT TR0
/(430) V2261_DIFF_PRS_VALGT_ER +2 V2261_DIFF_PRS_HJ1  ; DIFFERANSE MELLOM AKTUELT SETP. OG VALGT SETP, HJ  DIFFERANSE MELLOM AKTUELT SETP. OG VALGT SETP
AND 927.01
-(410) V2261_AKTUELT_PRS V2261_DIFF_PRS_HJ1 V2261_AKTUELT_PRS  ; ', HJ  DIFFERANSE MELLOM AKTUELT SETP. OG VALGT SETP
LD TR0
AND 927.02
+(400) V2261_AKTUELT_PRS V2261_DIFF_PRS_HJ1 V2261_AKTUELT_PRS  ; ', HJ  DIFFERANSE MELLOM AKTUELT SETP. OG VALGT SETP
LD TR0
ANDNOT PGM504_IND_C24  ; VASK PAST22
@AND PAST22_FRA_RUNL_UT  ; FRA RUNDLOP TIL UYKJOERING
MOV(021) V2261_PRS_VALGT V2261_AKTUELT_PRS  ; '

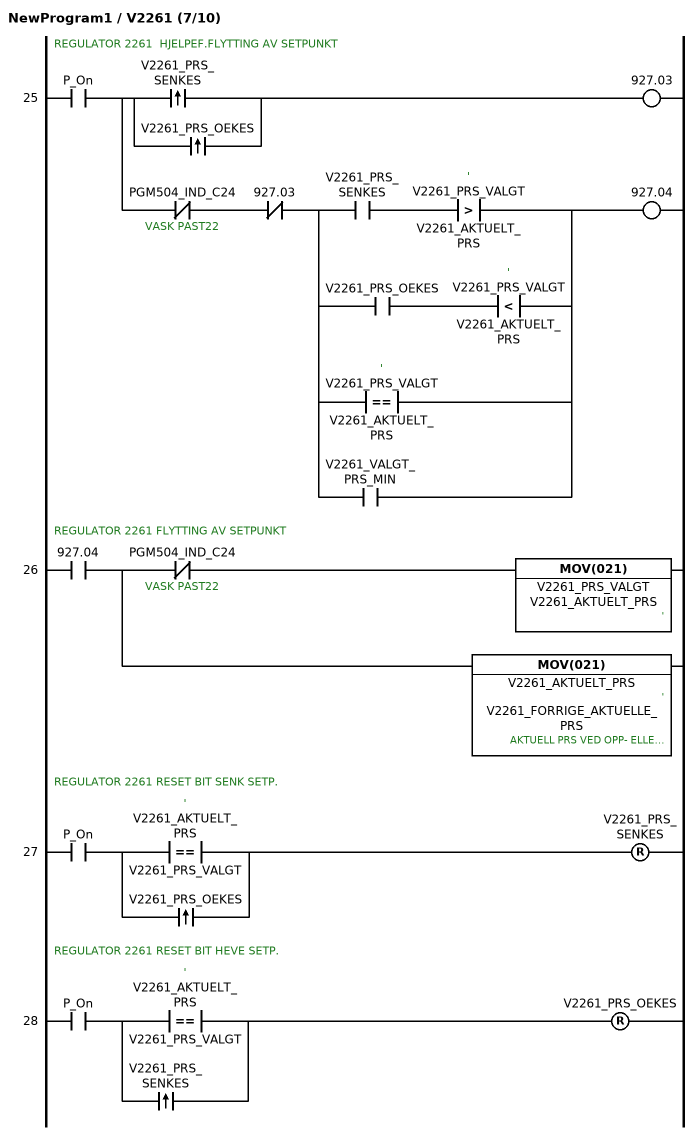
; rung 25: REGULATOR 2261  HJELPEF.FLYTTING AV SETPUNKT
LD P_On
OUT TR0
@LD V2261_PRS_SENKES
@OR V2261_PRS_OEKES
ANDLD
OUT 927.03
LD TR0
ANDNOT PGM504_IND_C24  ; VASK PAST22
ANDNOT 927.03
LD V2261_PRS_SENKES
AND>(320) V2261_PRS_VALGT V2261_AKTUELT_PRS  ; '
LD V2261_PRS_OEKES
AND<(310) V2261_PRS_VALGT V2261_AKTUELT_PRS  ; '
ORLD
OR=(300) V2261_PRS_VALGT V2261_AKTUELT_PRS  ; '
OR V2261_VALGT_PRS_MIN
ANDLD
OUT 927.04
; rung 26: REGULATOR 2261 FLYTTING AV SETPUNKT
LD 927.04
OUT TR0
ANDNOT PGM504_IND_C24  ; VASK PAST22
MOV(021) V2261_PRS_VALGT V2261_AKTUELT_PRS  ; '
LD TR0
MOV(021) V2261_AKTUELT_PRS V2261_FORRIGE_AKTUELLE_PRS  ; ', AKTUELL PRS VED OPP- ELLER NEDTRAPPING
; rung 27: REGULATOR 2261 RESET BIT SENK SETP.
LD P_On
LD=(300) V2261_AKTUELT_PRS V2261_PRS_VALGT  ; '
@OR V2261_PRS_OEKES
ANDLD
RSET V2261_PRS_SENKES
; rung 28: REGULATOR 2261 RESET BIT HEVE SETP.
LD P_On
LD=(300) V2261_AKTUELT_PRS V2261_PRS_VALGT  ; '
@OR V2261_PRS_SENKES
ANDLD
RSET V2261_PRS_OEKES

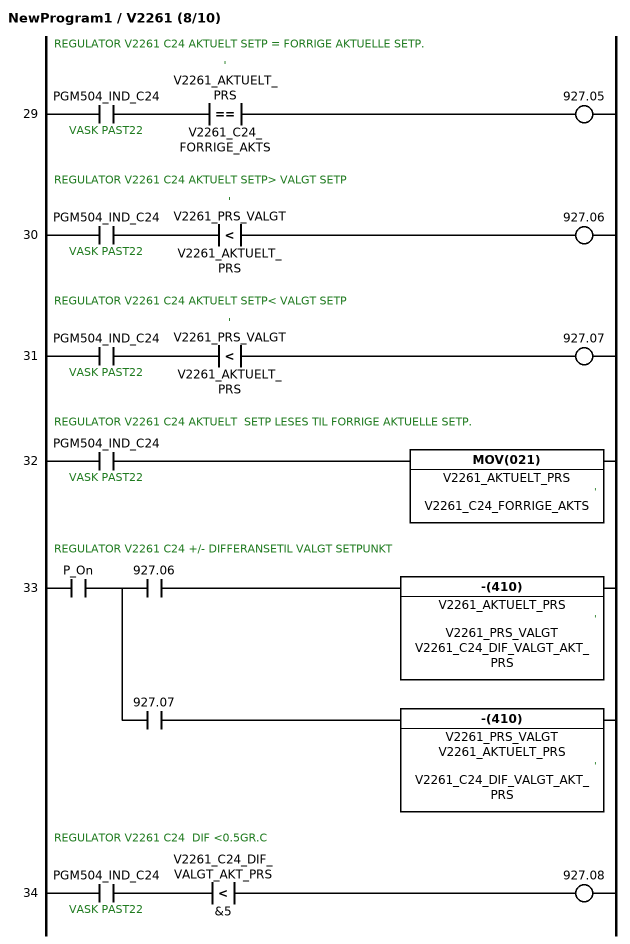
; rung 29: REGULATOR V2261 C24 AKTUELT SETP = FORRIGE AKTUELLE SETP.
LD PGM504_IND_C24  ; VASK PAST22
AND=(300) V2261_AKTUELT_PRS V2261_C24_FORRIGE_AKTS  ; '
OUT 927.05
; rung 30: REGULATOR V2261 C24 AKTUELT SETP> VALGT SETP
LD PGM504_IND_C24  ; VASK PAST22
AND<(310) V2261_PRS_VALGT V2261_AKTUELT_PRS  ; '
OUT 927.06
; rung 31: REGULATOR V2261 C24 AKTUELT SETP< VALGT SETP
LD PGM504_IND_C24  ; VASK PAST22
AND<(310) V2261_PRS_VALGT V2261_AKTUELT_PRS  ; '
OUT 927.07
; rung 32: REGULATOR V2261 C24 AKTUELT  SETP LESES TIL FORRIGE AKTUELLE SETP.
LD PGM504_IND_C24  ; VASK PAST22
MOV(021) V2261_AKTUELT_PRS V2261_C24_FORRIGE_AKTS  ; '
; rung 33: REGULATOR V2261 C24 +/- DIFFERANSETIL VALGT SETPUNKT
LD P_On
OUT TR0
AND 927.06
-(410) V2261_AKTUELT_PRS V2261_PRS_VALGT V2261_C24_DIF_VALGT_AKT_PRS  ; '
LD TR0
AND 927.07
-(410) V2261_PRS_VALGT V2261_AKTUELT_PRS V2261_C24_DIF_VALGT_AKT_PRS  ; '
; rung 34: REGULATOR V2261 C24  DIF <0.5GR.C
LD PGM504_IND_C24  ; VASK PAST22
AND<(310) V2261_C24_DIF_VALGT_AKT_PRS &5
OUT 927.08

